FUNCTION FUN_GetTime : STRING
VAR_INPUT
	stNtTime		:TIMESTRUCT;
END_VAR
VAR
	sTimestamp		:STRING;
END_VAR

// Add hour to timestamp
sTimestamp := '';
IF stNtTime.wHour < 10 THEN
	sTimestamp := CONCAT(sTimestamp,CONCAT('0', UINT_TO_STRING(stNtTime.wHour)));
ELSE
	sTimestamp := CONCAT(sTimestamp,UINT_TO_STRING(stNtTime.wHour));
END_IF

// Add min to timestamp
sTimestamp := CONCAT(sTimestamp, ':');
IF stNtTime.wMinute < 10 THEN
	sTimestamp := CONCAT(sTimestamp,CONCAT('0', UINT_TO_STRING(stNtTime.wMinute)));
ELSE
	sTimestamp := CONCAT(sTimestamp,UINT_TO_STRING(stNtTime.wMinute));
END_IF
sTimestamp := CONCAT(sTimestamp, ':');

// Add sec to timestamp
IF stNtTime.wSecond < 10 THEN
	sTimestamp := CONCAT(sTimestamp,CONCAT('0', UINT_TO_STRING(stNtTime.wSecond)));
ELSE
	sTimestamp := CONCAT(sTimestamp,UINT_TO_STRING(stNtTime.wSecond));
END_IF

// Return time
FUN_GetTime := sTimestamp;

END_FUNCTION

(* stored: Version 1.1.0.1, ProductVersion 3.1.4024.12
   POU FUN_GetTime: Id {b63e8ad1-effa-4ffe-8d96-a16a0373355e}, SpecialFunc None *)
